PROGRAM MAIN
VAR
	nastro : fb_msf();
	GVL_IO: INT;
END_VAR

nastro(
	start:= IO.start,
	stop:= IO.stop, 
	emg:= IO.emg, 
	ack:= IO.ack, 
	fc1:= IO.fc1, 
	fc2:= IO.fc2, 
	H1=> IO.H1, 
	HEMG=> IO.HEMG, 
	M=> IO.M,
	libero=>IO.libero
		);

END_PROGRAM

(* stored: Version 1.1.0.1, ProductVersion 3.1.4024.12
   POU MAIN: Id {5822dc26-d632-473a-86be-1f8ee9c088d2}, SpecialFunc None *)
